// TIA Portal V15.1 export
// export: Created 2024-05-17T05:38:13.916273Z, ExportSetting WithDefaults, DisplayName Totally Integrated Automation Portal, DisplayVersion V15.1 Update 5, DisplayName TIA Portal Openness, DisplayVersion V15.1 Update 5, DisplayName SINAMICS Startdrive Advanced, DisplayVersion V15.1, DisplayName G130, G150, S120, S150, SINAMICS MV, S210, DisplayVersion V15.1, DisplayName G110M, G120, G120C, G120D, G120P, DisplayVersion V15.1, DisplayName STEP 7 Professional, DisplayVersion V15.1 Update 5, DisplayName STEP 7 Safety, DisplayVersion V15.1, DisplayName WinCC Professional, DisplayVersion V15.1 Update 5, DisplayName SIMATIC Visualization Architect, DisplayVersion V15.1
DATA_BLOCK "_209210ZS01Safety"   // DB325
{ S7_Optimized_Access := 'FALSE' }
VERSION : 0.1
// stored: AutoNumber false, DBAccessibleFromOPCUA true, IsOnlyStoredInLoadMemory false, IsWriteProtectedInAS false
   VAR RETAIN
      AA_209210AS10F9SH1 { ExternalAccessible := 'False'; ExternalVisible := 'False'; ExternalWritable := 'False'} : Bool;   // Emergency Stop push button 210AS10 (Operator panel)
      AA_209210AS11F9SH1 { ExternalAccessible := 'False'; ExternalVisible := 'False'; ExternalWritable := 'False'} : Bool;   // Emergency Stop push button 210AS11 (Operator panel)
      AA_209210AS20F9SH1 { ExternalAccessible := 'False'; ExternalVisible := 'False'; ExternalWritable := 'False'} : Bool;   // Emergency Stop push button 210AS20 (Start/Stop panel)
      AA_209210AS40F9SH1 { ExternalAccessible := 'False'; ExternalVisible := 'False'; ExternalWritable := 'False'} : Bool;   // Emergency Stop push button 210AS40 (External panel)
      AA_209210AS41F9SH1 { ExternalAccessible := 'False'; ExternalVisible := 'False'; ExternalWritable := 'False'} : Bool;   // Emergency Stop push button 210AS41 (External panel)
      AA_209210ASH01F9SH1 { ExternalAccessible := 'False'; ExternalVisible := 'False'; ExternalWritable := 'False'} : Bool;   // Emergency Stop push button 210ASH01 (Handheld panel)
      AA_209210ASH01F9SH2 { ExternalAccessible := 'False'; ExternalVisible := 'False'; ExternalWritable := 'False'} : Bool;   // Deathmans switch 210ASH01 (Handheld panel)
      AA_209000AK03F9QC1FB { ExternalAccessible := 'False'; ExternalVisible := 'False'; ExternalWritable := 'False'} : Bool;   // Feedback Alarm Contactor Brake 400VAC OFF 210CR21
      AA_209000AK03F9QC2FB { ExternalAccessible := 'False'; ExternalVisible := 'False'; ExternalWritable := 'False'} : Bool;   // Feedback Alarm Contactor Brake 400VAC OFF 210CR21
      AA_209000AK03F9QC3FB { ExternalAccessible := 'False'; ExternalVisible := 'False'; ExternalWritable := 'False'} : Bool;   // Feedback Alarm Contactor Brake 400VAC OFF 210CS22
      AA_209000AK03F9QC4FB { ExternalAccessible := 'False'; ExternalVisible := 'False'; ExternalWritable := 'False'} : Bool;   // Feedback Alarm Contactor Brake 400VAC OFF 210CS22
      AA_209000AK03F9QC5FB { ExternalAccessible := 'False'; ExternalVisible := 'False'; ExternalWritable := 'False'} : Bool;   // Feedback Alarm Contactor Brake 400VAC OFF 210CR23
      AA_209000AK03F9QC6FB { ExternalAccessible := 'False'; ExternalVisible := 'False'; ExternalWritable := 'False'} : Bool;   // Feedback Alarm Contactor Brake 400VAC OFF 210CR23
      AA_209210AS20XS10 { ExternalAccessible := 'False'; ExternalVisible := 'False'; ExternalWritable := 'False'} : Bool;   // Dummy plug is missing, no Handheld is connected 210AS20 (Start/Stop panel)
      AC_209210CS22M4SG10F { ExternalAccessible := 'False'; ExternalVisible := 'False'; ExternalWritable := 'False'} : Bool;   // Body present buth the safety sensor is not activated 210CS22M410F
      AC_209210CS22M4SG11F { ExternalAccessible := 'False'; ExternalVisible := 'False'; ExternalWritable := 'False'} : Bool;   // Body present buth the safety sensor is not activated 210CS22M411F
      "AC_209000AK03M1-UE130PSC-1" { ExternalAccessible := 'False'; ExternalVisible := 'False'; ExternalWritable := 'False'} : Bool;   // Position speed control - The infeed roller is busy with a tranfer to the slat conveyor but the slat conveyor is not running/too slow
      "AC_209000AK03M4-UE131PSC-1" { ExternalAccessible := 'False'; ExternalVisible := 'False'; ExternalWritable := 'False'} : Bool;   // Position speed control - The slat conveyor is busy with a tranfer to the outfeed roller but the outfeed roller is not running/too slow
      AA_209210ZS01SafetNotReseted { ExternalAccessible := 'False'; ExternalVisible := 'False'; ExternalWritable := 'False'} : Bool;   // Safety not Reseted 210ZS01
      AD_209210ZS01EmergencyStop { ExternalAccessible := 'False'; ExternalVisible := 'False'; ExternalWritable := 'False'} : Bool;   // Emergency Stop 210ZS01
      AD_209210ZS01GateStop { ExternalAccessible := 'False'; ExternalVisible := 'False'; ExternalWritable := 'False'} : Bool;   // Gate Stop 210ZS01
      AD_209210ZS01FbkError { ExternalAccessible := 'False'; ExternalVisible := 'False'; ExternalWritable := 'False'} : Bool;   // Feedback Error Pilz/Contactor 210ZS01
      AD_209210ZS01EStopPLC212 { ExternalAccessible := 'False'; ExternalVisible := 'False'; ExternalWritable := 'False'} : Bool;   // Emergency Stop from PLC212
      AD_209210ZS01MStopPLC212 { ExternalAccessible := 'False'; ExternalVisible := 'False'; ExternalWritable := 'False'} : Bool;   // Motion Stop from PLC212 for roller 210CR23 & 210CS22
      AD_209210ZS01EStopPLC308 { ExternalAccessible := 'False'; ExternalVisible := 'False'; ExternalWritable := 'False'} : Bool;   // Emergency Stop from PLC318
      AD_209210ZS01MStopPLC308 { ExternalAccessible := 'False'; ExternalVisible := 'False'; ExternalWritable := 'False'} : Bool;   // Motion Stop from PLC318 for roller 210CR21
      "210AS10F9SH1AlarmABCondition" { ExternalAccessible := 'False'; ExternalVisible := 'False'; ExternalWritable := 'False'} : Bool;   // Alarm AB Condition
      "210AS11F9SH1AlarmABCondition" { ExternalAccessible := 'False'; ExternalVisible := 'False'; ExternalWritable := 'False'} : Bool;   // Alarm AB Condition
      "210AS20F9SH1AlarmABCondition" { ExternalAccessible := 'False'; ExternalVisible := 'False'; ExternalWritable := 'False'} : Bool;   // Alarm AB Condition
      "210AS40F9SH1AlarmABCondition" { ExternalAccessible := 'False'; ExternalVisible := 'False'; ExternalWritable := 'False'} : Bool;   // Alarm AB Condition
      "210AS41F9SH1AlarmABCondition" { ExternalAccessible := 'False'; ExternalVisible := 'False'; ExternalWritable := 'False'} : Bool;   // Alarm AB Condition
      "210ASH01F9SH1AlarmABCondition" { ExternalAccessible := 'False'; ExternalVisible := 'False'; ExternalWritable := 'False'} : Bool;   // Alarm AB Condition
      "210ASH01F9SH2AlarmABCondition" { ExternalAccessible := 'False'; ExternalVisible := 'False'; ExternalWritable := 'False'} : Bool;   // Alarm AB Condition
      "210AS20XS10AlarmABCondition" { ExternalAccessible := 'False'; ExternalVisible := 'False'; ExternalWritable := 'False'} : Bool;   // Alarm AB Condition
      AK03F9QC1FBAlarmABCondition { ExternalAccessible := 'False'; ExternalVisible := 'False'; ExternalWritable := 'False'} : Bool;   // Alarm AB Condition
      AK03F9QC2FBAlarmABCondition { ExternalAccessible := 'False'; ExternalVisible := 'False'; ExternalWritable := 'False'} : Bool;   // Alarm AB Condition
      AK03F9QC3FBAlarmABCondition { ExternalAccessible := 'False'; ExternalVisible := 'False'; ExternalWritable := 'False'} : Bool;   // Alarm AB Condition
      AK03F9QC4FBAlarmABCondition { ExternalAccessible := 'False'; ExternalVisible := 'False'; ExternalWritable := 'False'} : Bool;   // Alarm AB Condition
      AK03F9QC5FBAlarmABCondition { ExternalAccessible := 'False'; ExternalVisible := 'False'; ExternalWritable := 'False'} : Bool;   // Alarm AB Condition
      AK03F9QC6FBAlarmABCondition { ExternalAccessible := 'False'; ExternalVisible := 'False'; ExternalWritable := 'False'} : Bool;   // Alarm AB Condition
      SafetyNotResetedAlarmABCondition { ExternalAccessible := 'False'; ExternalVisible := 'False'; ExternalWritable := 'False'} : Bool;   // Alarm AB Condition
      H_209210AS10F9SH1IAnim : Word;   // Icon Animation
      H_209210AS11F9SH1IAnim : Word;   // Icon Animation
      H_209210AS20F9SH1IAnim : Word;   // Icon Animation
      H_209210AS40F9SH1IAnim : Word;   // Icon Animation
      H_209210AS41F9SH1IAnim : Word;   // Icon Animation
      H_209210ASH01F9SH1IAnim : Word;   // Icon Animation
      H_209210ASH01F9SH2IAnim : Word;   // Icon Animation
      H_209000AK03F9QC1FBIAnim : Word;   // Icon Animation
      H_209000AK03F9QC2FBIAnim : Word;   // Icon Animation
      H_209000AK03F9QC3FBIAnim : Word;   // Icon Animation
      H_209000AK03F9QC4FBIAnim : Word;   // Icon Animation
      H_209000AK03F9QC5FBIAnim : Word;   // Icon Animation
      H_209000AK03F9QC6FBIAnim : Word;   // Icon Animation
      H_209210AS20XS10IAnim : Word;   // Icon Animation
      H_209210CHB21M14SG1FIAnim : Word;   // Icon Animation
      H_209210CS22M4SG10FIAnim : Word;   // Icon Animation
      H_209210CS22M4SG11FIAnim : Word;   // Icon Animation
      H_209210ZS01SafetyNotResetedIAnim : Word;   // Icon Animation
      H_209210ZS01GateStopIAnim : Word;   // Icon Animation
      H_209210ZS01EmergencyStopIAnim : Word;   // Icon Animation
      H_209210ZS01FbkErrorIAnim : Word;   // Icon Animation
      H_209210ZS01EStopPLC212IAnim : Word;   // Icon Animation
      H_209210ZS01MStopPLC212IAnim : Word;   // Icon Animation
      H_209210ZS01EStopPLC308IAnim : Word;   // Icon Animation
      H_209210ZS01MStopPLC308IAnim : Word;   // Icon Animation
      H_209210ZS01PassivIAnim : Word;   // Icon Animation
      H_Anim : Word;   // Animation
      H_DBnr : Int;   // DB number
      Passivation { ExternalAccessible := 'False'; ExternalVisible := 'False'; ExternalWritable := 'False'} : "AlarmBits";   // Passivation Alarm Bits / Alarm A
      AlarmA { ExternalAccessible := 'False'; ExternalVisible := 'False'; ExternalWritable := 'False'} : Bool;   // Alarm A
      AlarmB { ExternalAccessible := 'False'; ExternalVisible := 'False'; ExternalWritable := 'False'} : Bool;   // Alarm B
      AlarmC { ExternalAccessible := 'False'; ExternalVisible := 'False'; ExternalWritable := 'False'} : Bool;   // Alarm C
      AlarmD { ExternalAccessible := 'False'; ExternalVisible := 'False'; ExternalWritable := 'False'} : Bool;   // Alarm D
      AlarmABCondition { ExternalAccessible := 'False'; ExternalVisible := 'False'; ExternalWritable := 'False'} : Bool;   // Summary Alarm AB condition
      SafetyObjectAckReq210AS10 { ExternalAccessible := 'False'; ExternalVisible := 'False'; ExternalWritable := 'False'} : Bool;   // Safety Status ACK REQ
      SafetyObjectAckReq210AS11 { ExternalAccessible := 'False'; ExternalVisible := 'False'; ExternalWritable := 'False'} : Bool;   // Safety Status ACK REQ
      SafetyObjectAckReq210AS20 { ExternalAccessible := 'False'; ExternalVisible := 'False'; ExternalWritable := 'False'} : Bool;   // Safety Status ACK REQ
      SafetyObjectAckReq210AS40 { ExternalAccessible := 'False'; ExternalVisible := 'False'; ExternalWritable := 'False'} : Bool;   // Safety Status ACK REQ
      SafetyObjectAckReq210AS41 { ExternalAccessible := 'False'; ExternalVisible := 'False'; ExternalWritable := 'False'} : Bool;   // Safety Status ACK REQ
      SafetyObjectAckReq210ASH01 { ExternalAccessible := 'False'; ExternalVisible := 'False'; ExternalWritable := 'False'} : Bool;   // Safety Status ACK REQ
      PowerOnRequest { ExternalAccessible := 'False'; ExternalVisible := 'False'; ExternalWritable := 'False'} : Bool;   // Power On Request
      ResetSafetyActive { ExternalAccessible := 'False'; ExternalVisible := 'False'; ExternalWritable := 'False'} : Bool;   // Reset Safety Active
      FeedbackError { ExternalAccessible := 'False'; ExternalVisible := 'False'; ExternalWritable := 'False'} : Bool;   // Feedback Error
      Check210CS22M4SG10F { ExternalAccessible := 'False'; ExternalVisible := 'False'; ExternalWritable := 'False'} : Bool;   // Check if both safety sensors are activated
      Check210AS20XS10 { ExternalAccessible := 'False'; ExternalVisible := 'False'; ExternalWritable := 'False'} : Bool;   // Check if dummy plug is ok
   END_VAR
BEGIN
END_DATA_BLOCK
